FUNCTION_BLOCK FB_MotionAxisNC IMPLEMENTS I_MotionAxis
VAR
    iHome : I_Home;
    iHalt : I_Halt;
    iPower : I_Power;
    iReset : I_Reset;
    iMoveAbsolute : I_MoveAbsolute;
    iReadParameter : I_ReadParameter;
    iWriteParameter  : I_WriteParameter;
    iParamSaveRestore: I_ParamSaveRestore;
    iEncoderScaling : I_EncoderScaling;
    iAxisStatus : I_AxisStatus;
    iBacklashCompensation : I_BacklashCompensation;
	{attribute 'hide'}
    bError: BOOL;
	{attribute 'hide'}
    nErrorID: UDINT;
	{attribute 'hide'}
    sMessage : T_MAXSTRING;
	{attribute 'hide'}
    rtAbortDone : R_TRIG;
	{attribute 'hide'}
    stMotionAxisStatus : ST_MotionAxisStatus;
END_VAR


ErrorHandling();

// update Motion Axis Outputs
stMotionAxisStatus.bAbortDone := iHalt.Done OR iReset.Done;
stMotionAxisStatus.bABorted := iMoveAbsolute.Aborted;
stMotionAxisStatus.bAxisEnable:=iAxisStatus.AxisEnabled();
stMotionAxisStatus.bAxisReadParamsInit := iReadParameter.AxisReadParamsInit;
stMotionAxisStatus.eAxisState := iAxisStatus.AxisState;
stMotionAxisStatus.bBacklashCompensationStatus := iBacklashCompensation.Status;
stMotionAxisStatus.bHaltActive := iHalt.Active;
stMotionAxisStatus.bHaltBusy := iHalt.Busy;
stMotionAxisStatus.bHaltDone := iHalt.Done;
stMotionAxisStatus.bHomeBusy := iHome.Busy;
stMotionAxisStatus.bHomeDone := iHome.Done;
stMotionAxisStatus.eHomeMode := iHome.Mode;
stMotionAxisStatus.bInTargetPosition := iAxisStatus.Done;
stMotionAxisStatus.nAxisId := iAxisStatus.AxisID;
stMotionAxisStatus.fMeasuredAcceleration := iAxisStatus.MeasuredAcceleration;
stMotionAxisStatus.fMeasuredCompensation := iBacklashCompensation.CurrentBacklash;
stMotionAxisStatus.fMeasuredPosition := iAxisStatus.MeasuredPosition;
stMotionAxisStatus.fMeasuredPositionDiff := iAxisStatus.MeasuredPositionDiff;
stMotionAxisStatus.fMeasuredVelocity := iAxisStatus.MeasuredVelocity;
stMotionAxisStatus.sMessage :=sMessage;
stMotionAxisStatus.bMoveAbsoluteAborted := iMoveAbsolute.Aborted;
stMotionAxisStatus.bMoveAbsoluteActive := iMoveAbsolute.Active;
stMotionAxisStatus.bMoveAbsoluteBusy := iMoveAbsolute.Busy;
stMotionAxisStatus.bMoveAbsoluteDone := iMoveAbsolute.Done;
stMotionAxisStatus.bNegativeMotionIsEnabled := iAxisStatus.NegativeMotionIsEnabled;
stMotionAxisStatus.bPositiveMotionIsEnabled := iAxisStatus.PositiveMotionIsEnabled;
stMotionAxisStatus.bPowerActive := iPower.PowerIsEnabled;
stMotionAxisStatus.fPowerOverride := iPower.Override;
stMotionAxisStatus.bResetBusy := iReset.Busy;
stMotionAxisStatus.bResetDone := iReset.Done;
stMotionAxisStatus.fSavedPosition := iParamSaveRestore.SavedPosition;
stMotionAxisStatus.nScaledEncoderCount := iEncoderScaling.EncoderCount;
stMotionAxisStatus.bStandStill := iAxisStatus.StandStill;
stMotionAxisStatus.bBusy := iHome.Busy OR iMoveAbsolute.Busy;
stMotionAxisStatus.bDone := iHome.Done OR iMoveAbsolute.Done;
stMotionAxisStatus.bError := bError;
stMotionAxisStatus.nErrorID := nErrorID;

METHOD AxisEnabled : BOOL
VAR_INPUT
END_VAR
AxisEnabled:=THIS^.iAxisStatus.AxisEnabled();
END_METHOD

(*
    Handle positive/negative backlash compensation
    User needs to set the direction of backlash from the sign of the compensation value
    Backlash compensation is disabled during referencing (homing).
    When direction is positive/negative, further movement in the negative/positive direction not compensated
    further movement in the negative/positive direction will be compensated
*)
METHOD BacklashCompensation
VAR_INPUT
	Enable : BOOL := FALSE;
	RampVelo : LREAL;
END_VAR
THIS^.iBacklashCompensation.BacklashCompensation(	Enable:=Enable,
													RampVelo:=RampVelo
                                                );
END_METHOD

METHOD PUBLIC CallAfterInit
VAR_INPUT
    iHome : I_Home;
    iHalt : I_Halt;
    iPower : I_Power;
    iReset : I_Reset;
    iMoveAbsolute : I_MoveAbsolute;
    iReadParameter : I_ReadParameter;
    iWriteParameter  : I_WriteParameter;
    iParamSaveRestore: I_ParamSaveRestore;
    iEncoderScaling : I_EncoderScaling;
    iAxisStatus : I_AxisStatus;
    iBacklashCompensation : I_BacklashCompensation;
END_VAR
THIS^.iHome := iHome;
THIS^.iHalt := iHalt;
THIS^.iPower := iPower;
THIS^.iReset := iReset;
THIS^.iMoveAbsolute := iMoveAbsolute;
THIS^.iReadParameter := iReadParameter ;
THIS^.iWriteParameter  := iWriteParameter;
THIS^.iParamSaveRestore:= iParamSaveRestore;
THIS^.iEncoderScaling := iEncoderScaling;
THIS^.iAxisStatus := iAxisStatus;
THIS^.iBacklashCompensation  := iBacklashCompensation ;
END_METHOD

METHOD DisablePower
THIS^.iPower.DisablePower();
END_METHOD

METHOD DriveCommands
VAR_INPUT
    HomeCmd	: BOOL;
    NewMoveReq	: BOOL;
    EnableMode	: E_StageEnableMode;
END_VAR
END_METHOD

METHOD ErrorHandling
(*
    Error from NC functions
    The error will be sent to EPICS interface based on predifined
    priority: axis, power, backlash, absoluteMove, etc...
*)
IF THIS^.iPower.Error AND THIS^.iPower.PowerIsEnabled THEN
    bError:=THIS^.iPower.Error;
    nErrorId:=THIS^.iPower.ErrorID;
    sMessage := THIS^.iPower.Message;
ELSIF THIS^.iHalt.Error AND THIS^.iHalt.Active THEN
    bError:=THIS^.iHalt.Error;
    nErrorId:=THIS^.iHalt.ErrorID;
    sMessage := THIS^.iHalt.Message;
ELSIF THIS^.iReset.Error AND THIS^.iReset.Active THEN
    bError:=THIS^.iReset.Error;
    nErrorId:=THIS^.iReset.ErrorID;
    sMessage := THIS^.iReset.Message;
ELSIF THIS^.iBacklashCompensation.Error THEN
    bError:=THIS^.iBacklashCompensation.Error;
    nErrorId:=THIS^.iBacklashCompensation.ErrorID;
    sMessage := THIS^.iBacklashCompensation.Message;
ELSIF THIS^.iMoveAbsolute.Error THEN
    bError:=THIS^.iMoveAbsolute.Error;
    nErrorId:=THIS^.iMoveAbsolute.ErrorID;
    sMessage := THIS^.iMoveAbsolute.Message;
ELSIF THIS^.iHome.Error (*Homing error*) THEN
    bError:=THIS^.iHome.Error;
    nErrorId:=THIS^.iHome.ErrorID;
    sMessage := THIS^.iHome.Message;
ELSIF THIS^.iAxisStatus.Error  THEN
    bError:=THIS^.iAxisStatus.Error;
    nErrorId:=THIS^.iAxisStatus.ErrorID;
    sMessage := THIS^.iAxisStatus.Message;
ELSIF THIS^.iReadParameter.Error THEN
    bError := THIS^.iReadParameter.Error;
    nErrorId := THIS^.iReadParameter.ErrorID;
    sMessage := THIS^.iReadParameter.Message;
ELSIF THIS^.iWriteParameter.Error THEN
    bError := THIS^.iWriteParameter.Error;
    nErrorId := THIS^.iWriteParameter.ErrorID;
    sMessage := THIS^.iWriteParameter.Message;
ELSIF THIS^.iParamSaveRestore.Error THEN
    bError := THIS^.iParamSaveRestore.Error;
    nErrorId := THIS^.iParamSaveRestore.ErrorID;
    sMessage := THIS^.iParamSaveRestore.Message;
ELSE
    bError:=FALSE;
    nErrorId:=0;
    sMessage := '';
END_IF;
END_METHOD

//FB_Init is always available implicitly and it is used primarily for initialization.
//The return value is not evaluated. For a specific influence, you can also declare the
//methods explicitly and provide additional code there with the standard initialization
//code. You can evaluate the return value.
METHOD FB_Init: BOOL
VAR_INPUT
    bInitRetains: BOOL; // TRUE: the retain variables are initialized (reset warm / reset cold)
    bInCopyCode: BOOL;  // TRUE: the instance will be copied to the copy code afterward (online change)

    iHome : I_Home;
    iHalt : I_Halt;
    iPower : I_Power;
    iReset : I_Reset;
    iMoveAbsolute : I_MoveAbsolute;
    iReadParameter : I_ReadParameter;
    iWriteParameter  : I_WriteParameter;
    iParamSaveRestore: I_ParamSaveRestore;
    iEncoderScaling : I_EncoderScaling;
    iAxisStatus : I_AxisStatus;
    iBacklashCompensation : I_BacklashCompensation;
END_VAR
THIS^.iHome := iHome;
THIS^.iHalt := iHalt;
THIS^.iPower := iPower;
THIS^.iReset := iReset;
THIS^.iMoveAbsolute := iMoveAbsolute;
THIS^.iReadParameter := iReadParameter ;
THIS^.iWriteParameter  := iWriteParameter;
THIS^.iParamSaveRestore:= iParamSaveRestore;
THIS^.iEncoderScaling := iEncoderScaling;
THIS^.iAxisStatus := iAxisStatus;
THIS^.iBacklashCompensation  := iBacklashCompensation ;
END_METHOD

METHOD Halt
VAR_INPUT
    Deceleration	: LREAL := 0;
    Jerk	: LREAL := 0;
    BufferMode	: MC_BufferMode := MC_BufferMode.MC_Aborting;
END_VAR
THIS^.iHalt.Halt( 	Deceleration:=Deceleration,
                    Jerk:=Jerk ,
                    BufferMode:=BufferMode );
END_METHOD

METHOD Home
VAR_INPUT
    Position        : LREAL         := DEFAULT_HOME_POSITION;
    BufferMode      : MC_BufferMode;
END_VAR
//
THIS^.iHome.Home(Position:=0.0,BufferMode:=MC_BufferMode.MC_Aborting);
END_METHOD

METHOD MoveAbsolute
VAR_INPUT
    Position	: LREAL;
    Velocity	: LREAL;
    Acceleration	: LREAL := 0.0;
    Deceleration	: LREAL := 0.0;
    Jerk	: LREAL := 0.0;
    BufferMode	: MC_BufferMode := MC_BufferMode.MC_Aborting;
END_VAR
THIS^.iMoveAbsolute.MoveAbsolute( 	Position:=Position,
                                       Velocity := Velocity,
                                    Acceleration := Acceleration,
                                    Deceleration := Deceleration,
                                    Jerk := Jerk,
                                    BufferMode := BufferMode);
END_METHOD

METHOD Power
VAR_INPUT
    Enable	: BOOL;
    Enable_Positive	: BOOL;
    Enable_Negative	: BOOL;
    Override	: LREAL := 100.0;
    BufferMode	: MC_BufferMode := MC_BufferMode.MC_Aborting;
END_VAR
THIS^.iPower.Power(	Enable:=Enable,
                    Enable_Positive:= Enable_Positive,
                    Enable_Negative:=Enable_Negative,
                    Override:=Override,
                    BufferMode:=BufferMode
                );
END_METHOD

(*This is overriden by this object internal acess to the interlock instance
  this is intended to pass power enable flags via the fbMotionDrive
*)
METHOD PowerEnables
VAR_INPUT
    Enable	: BOOL;
    Enable_Positive	: BOOL;
    Enable_Negative	: BOOL;
END_VAR
THIS^.iPower.Power(	Enable:=Enable,
                    Enable_Positive:= Enable_Positive,
                    Enable_Negative:=Enable_Negative,
                    Override:=100.0,
                    BufferMode:=MC_BufferMode.MC_Aborting
                );
END_METHOD

METHOD ReadAxisParams
VAR_INPUT
    Enable	: BOOL;
    RefreshDelay	: TIME;
END_VAR
THIS^.iReadParameter.ReadParameters(Enable:=Enable, RefreshDelay:=RefreshDelay);
END_METHOD

METHOD Reset
VAR_INPUT
END_VAR
THIS^.iReset.Reset();
END_METHOD

METHOD SaveAxisParams
VAR_INPUT
    Enable	: BOOL;
END_VAR
THIS^.iParamSaveRestore.SaveAxisParams(Enable:=Enable);
END_METHOD

PROPERTY Status : REFERENCE TO ST_MotionAxisStatus
GET
Status REF= stMotionAxisStatus;
END_GET
END_PROPERTY

END_FUNCTION_BLOCK

(* stored: Version 1.1.0.1
   POU FB_MotionAxisNC: Id {b2082997-3f19-4e96-8959-1acebaf0fbc0}, SpecialFunc None
   Method AxisEnabled: Id {cc4bbafd-6987-498c-9fa8-c674abc392f5}
   Method BacklashCompensation: Id {47b7a29c-5a46-4b34-82e5-46809c891caa}
   Method CallAfterInit: Id {9b35c028-bf1f-45b2-b785-efd534d69557}
   Method DisablePower: Id {d431613d-dd04-4413-bd5f-ff595b13e90c}
   Method DriveCommands: Id {b8507c31-2c0f-4ad7-a181-843fb8302b04}
   Method ErrorHandling: Id {47e04ad9-0158-4554-a680-9fdc3b3acad9}
   Method FB_Init: Id {3ca36ea2-2fee-4826-a4c8-a0afdd04a31e}
   Method Halt: Id {669b312b-74c8-481c-b6f9-68179672a70f}
   Method Home: Id {19a4a42c-65d0-44c2-9ba0-43e7fa25e791}
   Method MoveAbsolute: Id {4f09799f-35f4-498c-b47e-65f81ea0c180}
   Method Power: Id {ec1783df-e1a3-46f4-829a-9762b3ca588d}
   Method PowerEnables: Id {9f48c379-e1d3-4087-91db-594e6015e37d}
   Method ReadAxisParams: Id {050cbcc2-33e7-4ef4-8d73-511312ef4239}
   Method Reset: Id {1c7b54c7-fc14-4552-871c-6730dd93d7ea}
   Method SaveAxisParams: Id {e5a35223-1f28-40e0-a094-53d1b9164718}
   Property Status: Id {e57f34f0-4782-4fdb-b236-ad33acfccad4}
   Get Get: Id {19f70767-a91a-4512-8e71-3365cb03cfc5} *)
